{attribute 'qualified_only'}
VAR_GLOBAL
	// Digital IO in FactoryIO Outputs
	mb_Input_Coils		:	ARRAY [0..3] OF BOOL;
	// Digital IO in FactoryIO Inputs
	mb_Output_Coils		:   ARRAY [0..9] OF BOOL;
	// Analog IO in FactoryIO Outputs
	mb_Input_Registers	: 	ARRAY [0..2] OF WORD;
	// Analog IO in FactoryIO Inputs
	mb_Output_Registers	: 	ARRAY [0..1] OF WORD;
	
	nState				: INT;
END_VAR

(* stored: Version 1.1.0.1, ProductVersion 3.1.4024.12
   GVL GVL: Id {f5dc6345-1f38-4419-9302-b9eecfc8063c} *)
